FUNCTION_BLOCK Position IMPLEMENTS I_Position, I_PosStation
VAR_INPUT
END_VAR
VAR_OUTPUT
END_VAR
VAR
	_position		: LREAL;
	_enableRequest 	: BOOL;
	_IMover			: I_MoverPos;
	_requestStep 	: UDINT;
	_posID			: UDINT;
END_VAR

METHOD EnableRequest : BOOL
VAR_INPUT
	OnOff : BOOL;
END_VAR
_EnableRequest := OnOff;
EnableRequest := RequestMover;
END_METHOD

//FB_Init is always available implicitly and it is used primarily for initialization.
//The return value is not evaluated. For a specific influence, you can also declare the
//methods explicitly and provide additional code there with the standard initialization
//code. You can evaluate the return value.
METHOD FB_Init: BOOL
VAR_INPUT
    bInitRetains: BOOL; // TRUE: the retain variables are initialized (reset warm / reset cold)
    bInCopyCode: BOOL;  // TRUE: the instance will be copied to the copy code afterward (online change)
	position : LREAL;  
	manager : I_RegisterPosition; 
END_VAR
_position := position;
manager.RegisterPosition(THIS^);
END_METHOD

{warning 'Add property implementation'}
PROPERTY InPosition : BOOL
GET
VAR
	difference	: LREAL;
	tolerance 	: LREAL := 100;
END_VAR
IF _IMover <> 0 THEN
	difference := ABS(_position - _IMover.Position);
	IF difference < tolerance THEN
		InPosition := TRUE;
	END_IF	
END_IF
END_GET
END_PROPERTY

PROPERTY Linked : BOOL
GET
Linked := _IMover <> 0;
END_GET
END_PROPERTY

METHOD MoverChangeStep : BOOL
VAR_INPUT
	step	: UDINT;
END_VAR
IF _IMover <> 0 THEN
	_IMover.ChangeStep(step);
END_IF
END_METHOD

PROPERTY RequestedStep : UDINT
GET
RequestedStep := _requestStep;
END_GET
SET
_requestStep := RequestedStep;
END_SET
END_PROPERTY

{warning 'Add property implementation'}
PROPERTY RequestMover : BOOL
GET
IF _IMover <> 0 THEN
	_enableRequest := FALSE;
END_IF
RequestMover := _enableRequest;
END_GET
END_PROPERTY

METHOD SetAttractStep : BOOL
VAR_INPUT
	step	: INT;
END_VAR
_requestStep := step;
END_METHOD

METHOD SetMoverLink : BOOL
VAR_INPUT
	mover : I_MoverPos;
END_VAR
_IMover := mover;
END_METHOD

PROPERTY TargetPosition : LREAL
GET
TargetPosition := _position;
END_GET
END_PROPERTY

END_FUNCTION_BLOCK

(* stored: Version 1.1.0.1
   POU Position: Id {0640af27-2fc8-44fa-9165-1e7a19ffa04d}, SpecialFunc None
   Folder Constructor: Id {dddf045b-c3a5-46d1-8cc6-cb6803c75dcb}
   Method EnableRequest: Id {50846eb0-7075-4335-9ffc-b4c3c39d73de}
   Method FB_Init: Id {b2662626-7fd1-4ca5-b662-eee38d3e844e}
   Property InPosition: Id {2140a580-6154-4bdf-9b1e-ad5c95f4078c}
   Get Get: Id {38d390b9-7b5b-4697-8a64-0eee27c851fb}
   Property Linked: Id {68707e32-0222-48f9-8cab-195cae589404}
   Get Get: Id {e8e717ef-e0b2-4645-bab5-c1d06fd3fceb}
   Method MoverChangeStep: Id {9b4086f8-0788-46ff-994c-bcca2b222e8f}
   Property RequestedStep: Id {de5c08fa-11b8-4863-86c0-8cf94dc3b7ab}
   Get Get: Id {e50c3b44-0088-4672-b2ac-804db80a7b1f}
   Set Set: Id {cf40b16e-1a62-446d-93a9-a8429a7bd5a7}
   Property RequestMover: Id {7fa1da01-6b4b-47c2-9ce2-ac14f4c935f7}
   Get Get: Id {4694d44e-c646-4c9d-b1eb-b6b0461598cb}
   Method SetAttractStep: Id {f85949cf-0a35-4ace-9391-7b7cad52bd71}
   Method SetMoverLink: Id {c57b5a31-fd28-499d-87a1-775b14df67f1}
   Property TargetPosition: Id {942bd01f-5e5a-487d-9243-d7755b08ab84}
   Get Get: Id {45214525-edb3-4aea-bfed-c9fbc3ee2c2c} *)
